Yaskawa INFORM job: sDeep_drilling_(2).JBI

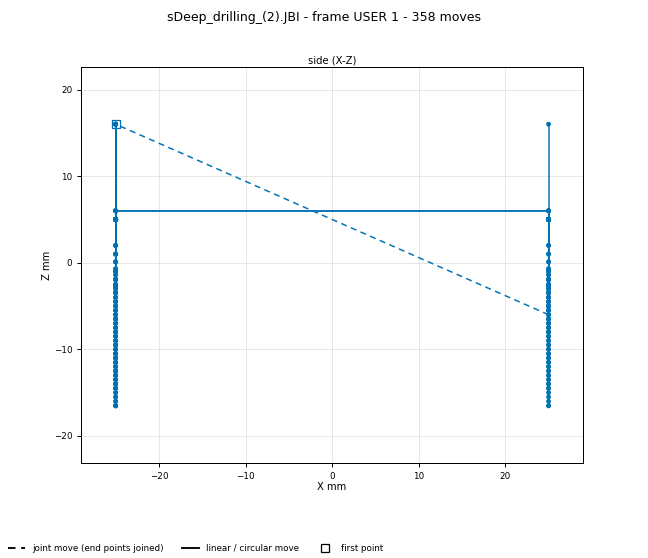
[picture p0: tool path of sDeep_drilling_(2).JBI in frame USER 1, 358 of 358 moves have a stored position in this frame; points joined in program order, loops and branches not executed]
/JOB
//NAME sDeep_drilling_(2)
//POS
///NPOS 194,0,0,0,0,0
///USER 1
///TOOL 3
///POSTYPE USER
///RECTAN
///RCONF 1,0,0,0,0,0
C00000=-25.000,10.000,16.000,0.000,-180.000,-30.000
C00001=-25.000,10.000,16.000,0.000,-180.000,-30.000
C00002=-25.000,10.000,6.000,0.000,-180.000,-30.000
C00003=-25.000,10.000,5.000,0.000,-180.000,-30.000
C00004=-25.000,10.000,-16.535,0.000,-180.000,-30.000
C00005=-25.000,10.000,6.000,0.000,-180.000,-30.000
C00006=25.000,10.000,6.000,0.000,-180.000,-30.000
C00007=25.000,10.000,6.000,0.000,-180.000,-30.000
C00008=25.000,10.000,5.000,0.000,-180.000,-30.000
C00009=25.000,10.000,-16.535,0.000,-180.000,-30.000
C00010=25.000,10.000,6.000,0.000,-180.000,-30.000
C00011=25.000,10.000,16.000,0.000,-180.000,-30.000
C00000=-25.000,10.000,16.000,0.000,-180.000,-30.000
C00001=-25.000,10.000,16.000,0.000,-180.000,-30.000
C00002=-25.000,10.000,6.000,0.000,-180.000,-30.000
C00003=-25.000,10.000,5.000,0.000,-180.000,-30.000
C00004=-25.000,10.000,-16.535,0.000,-180.000,-30.000
C00005=-25.000,10.000,6.000,0.000,-180.000,-30.000
C00006=25.000,10.000,6.000,0.000,-180.000,-30.000
C00007=25.000,10.000,6.000,0.000,-180.000,-30.000
C00008=25.000,10.000,5.000,0.000,-180.000,-30.000
C00009=25.000,10.000,-16.535,0.000,-180.000,-30.000
C00010=25.000,10.000,6.000,0.000,-180.000,-30.000
C00011=25.000,10.000,16.000,0.000,-180.000,-30.000
C00000=-25.000,10.000,16.000,0.000,-180.000,-30.000
C00001=-25.000,10.000,16.000,0.000,-180.000,-30.000
C00002=-25.000,10.000,6.000,0.000,-180.000,-30.000
C00003=-25.000,10.000,5.000,0.000,-180.000,-30.000
C00004=-25.000,10.000,2.000,0.000,-180.000,-30.000
C00005=-25.000,10.000,-1.000,0.000,-180.000,-30.000
C00006=-25.000,10.000,-0.898,0.000,-180.000,-30.000
C00007=-25.000,10.000,-1.900,0.000,-180.000,-30.000
C00008=-25.000,10.000,-1.798,0.000,-180.000,-30.000
C00009=-25.000,10.000,-2.700,0.000,-180.000,-30.000
C00010=-25.000,10.000,-2.598,0.000,-180.000,-30.000
C00011=-25.000,10.000,-3.400,0.000,-180.000,-30.000
C00012=-25.000,10.000,-3.298,0.000,-180.000,-30.000
C00013=-25.000,10.000,-4.000,0.000,-180.000,-30.000
C00014=-25.000,10.000,-3.898,0.000,-180.000,-30.000
C00015=-25.000,10.000,-4.500,0.000,-180.000,-30.000
C00016=-25.000,10.000,-4.398,0.000,-180.000,-30.000
C00017=-25.000,10.000,-5.000,0.000,-180.000,-30.000
C00018=-25.000,10.000,6.000,0.000,-180.000,-30.000
C00019=-25.000,10.000,-3.000,0.000,-180.000,-30.000
C00020=-25.000,10.000,-5.500,0.000,-180.000,-30.000
C00021=-25.000,10.000,-5.398,0.000,-180.000,-30.000
C00022=-25.000,10.000,-6.000,0.000,-180.000,-30.000
C00023=-25.000,10.000,-5.898,0.000,-180.000,-30.000
C00024=-25.000,10.000,-6.500,0.000,-180.000,-30.000
C00025=-25.000,10.000,-6.398,0.000,-180.000,-30.000
C00026=-25.000,10.000,-7.000,0.000,-180.000,-30.000
C00027=-25.000,10.000,-6.898,0.000,-180.000,-30.000
C00028=-25.000,10.000,-7.500,0.000,-180.000,-30.000
C00029=-25.000,10.000,-7.398,0.000,-180.000,-30.000
C00030=-25.000,10.000,-8.000,0.000,-180.000,-30.000
C00031=-25.000,10.000,-7.898,0.000,-180.000,-30.000
C00032=-25.000,10.000,-8.500,0.000,-180.000,-30.000
C00033=-25.000,10.000,-8.398,0.000,-180.000,-30.000
C00034=-25.000,10.000,-9.000,0.000,-180.000,-30.000
C00035=-25.000,10.000,-8.898,0.000,-180.000,-30.000
C00036=-25.000,10.000,-9.500,0.000,-180.000,-30.000
C00037=-25.000,10.000,-9.398,0.000,-180.000,-30.000
C00038=-25.000,10.000,-10.000,0.000,-180.000,-30.000
C00039=-25.000,10.000,6.000,0.000,-180.000,-30.000
C00040=-25.000,10.000,-8.000,0.000,-180.000,-30.000
C00041=-25.000,10.000,-10.500,0.000,-180.000,-30.000
C00042=-25.000,10.000,-10.398,0.000,-180.000,-30.000
C00043=-25.000,10.000,-11.000,0.000,-180.000,-30.000
C00044=-25.000,10.000,-10.898,0.000,-180.000,-30.000
C00045=-25.000,10.000,-11.500,0.000,-180.000,-30.000
C00046=-25.000,10.000,-11.398,0.000,-180.000,-30.000
C00047=-25.000,10.000,-12.000,0.000,-180.000,-30.000
C00048=-25.000,10.000,-11.898,0.000,-180.000,-30.000
C00049=-25.000,10.000,-12.500,0.000,-180.000,-30.000
C00050=-25.000,10.000,-12.398,0.000,-180.000,-30.000
C00051=-25.000,10.000,-13.000,0.000,-180.000,-30.000
C00052=-25.000,10.000,-12.898,0.000,-180.000,-30.000
C00053=-25.000,10.000,-13.500,0.000,-180.000,-30.000
C00054=-25.000,10.000,-13.398,0.000,-180.000,-30.000
C00055=-25.000,10.000,-14.000,0.000,-180.000,-30.000
C00056=-25.000,10.000,-13.898,0.000,-180.000,-30.000
C00057=-25.000,10.000,-14.500,0.000,-180.000,-30.000
C00058=-25.000,10.000,-14.398,0.000,-180.000,-30.000
C00059=-25.000,10.000,-15.000,0.000,-180.000,-30.000
C00060=-25.000,10.000,6.000,0.000,-180.000,-30.000
C00061=-25.000,10.000,-13.000,0.000,-180.000,-30.000
C00062=-25.000,10.000,-15.500,0.000,-180.000,-30.000
C00063=-25.000,10.000,-15.398,0.000,-180.000,-30.000
C00064=-25.000,10.000,-16.000,0.000,-180.000,-30.000
C00065=-25.000,10.000,-15.898,0.000,-180.000,-30.000
C00066=-25.000,10.000,-16.500,0.000,-180.000,-30.000
C00067=-25.000,10.000,-16.398,0.000,-180.000,-30.000
C00068=-25.000,10.000,-16.535,0.000,-180.000,-30.000
C00069=-25.000,10.000,6.000,0.000,-180.000,-30.000
C00070=25.000,10.000,6.000,0.000,-180.000,-30.000
C00071=25.000,10.000,6.000,0.000,-180.000,-30.000
C00072=25.000,10.000,5.000,0.000,-180.000,-30.000
C00073=25.000,10.000,2.000,0.000,-180.000,-30.000
C00074=25.000,10.000,-1.000,0.000,-180.000,-30.000
C00075=25.000,10.000,-0.898,0.000,-180.000,-30.000
C00076=25.000,10.000,-1.900,0.000,-180.000,-30.000
C00077=25.000,10.000,-1.798,0.000,-180.000,-30.000
C00078=25.000,10.000,-2.700,0.000,-180.000,-30.000
C00079=25.000,10.000,-2.598,0.000,-180.000,-30.000
C00080=25.000,10.000,-3.400,0.000,-180.000,-30.000
C00081=25.000,10.000,-3.298,0.000,-180.000,-30.000
C00082=25.000,10.000,-4.000,0.000,-180.000,-30.000
C00083=25.000,10.000,-3.898,0.000,-180.000,-30.000
C00084=25.000,10.000,-4.500,0.000,-180.000,-30.000
C00085=25.000,10.000,-4.398,0.000,-180.000,-30.000
C00086=25.000,10.000,-5.000,0.000,-180.000,-30.000
C00087=25.000,10.000,6.000,0.000,-180.000,-30.000
C00088=25.000,10.000,-3.000,0.000,-180.000,-30.000
C00089=25.000,10.000,-5.500,0.000,-180.000,-30.000
C00090=25.000,10.000,-5.398,0.000,-180.000,-30.000
C00091=25.000,10.000,-6.000,0.000,-180.000,-30.000
C00092=25.000,10.000,-5.898,0.000,-180.000,-30.000
C00093=25.000,10.000,-6.500,0.000,-180.000,-30.000
C00094=25.000,10.000,-6.398,0.000,-180.000,-30.000
C00095=25.000,10.000,-7.000,0.000,-180.000,-30.000
C00096=25.000,10.000,-6.898,0.000,-180.000,-30.000
C00097=25.000,10.000,-7.500,0.000,-180.000,-30.000
C00098=25.000,10.000,-7.398,0.000,-180.000,-30.000
C00099=25.000,10.000,-8.000,0.000,-180.000,-30.000
C00100=25.000,10.000,-7.898,0.000,-180.000,-30.000
C00101=25.000,10.000,-8.500,0.000,-180.000,-30.000
C00102=25.000,10.000,-8.398,0.000,-180.000,-30.000
C00103=25.000,10.000,-9.000,0.000,-180.000,-30.000
C00104=25.000,10.000,-8.898,0.000,-180.000,-30.000
C00105=25.000,10.000,-9.500,0.000,-180.000,-30.000
C00106=25.000,10.000,-9.398,0.000,-180.000,-30.000
C00107=25.000,10.000,-10.000,0.000,-180.000,-30.000
C00108=25.000,10.000,6.000,0.000,-180.000,-30.000
C00109=25.000,10.000,-8.000,0.000,-180.000,-30.000
C00110=25.000,10.000,-10.500,0.000,-180.000,-30.000
C00111=25.000,10.000,-10.398,0.000,-180.000,-30.000
C00112=25.000,10.000,-11.000,0.000,-180.000,-30.000
C00113=25.000,10.000,-10.898,0.000,-180.000,-30.000
C00114=25.000,10.000,-11.500,0.000,-180.000,-30.000
C00115=25.000,10.000,-11.398,0.000,-180.000,-30.000
C00116=25.000,10.000,-12.000,0.000,-180.000,-30.000
C00117=25.000,10.000,-11.898,0.000,-180.000,-30.000
C00118=25.000,10.000,-12.500,0.000,-180.000,-30.000
C00119=25.000,10.000,-12.398,0.000,-180.000,-30.000
C00120=25.000,10.000,-13.000,0.000,-180.000,-30.000
C00121=25.000,10.000,-12.898,0.000,-180.000,-30.000
C00122=25.000,10.000,-13.500,0.000,-180.000,-30.000
C00123=25.000,10.000,-13.398,0.000,-180.000,-30.000
C00124=25.000,10.000,-14.000,0.000,-180.000,-30.000
C00125=25.000,10.000,-13.898,0.000,-180.000,-30.000
C00126=25.000,10.000,-14.500,0.000,-180.000,-30.000
C00127=25.000,10.000,-14.398,0.000,-180.000,-30.000
C00128=25.000,10.000,-15.000,0.000,-180.000,-30.000
C00129=25.000,10.000,6.000,0.000,-180.000,-30.000
C00130=25.000,10.000,-13.000,0.000,-180.000,-30.000
C00131=25.000,10.000,-15.500,0.000,-180.000,-30.000
C00132=25.000,10.000,-15.398,0.000,-180.000,-30.000
C00133=25.000,10.000,-16.000,0.000,-180.000,-30.000
C00134=25.000,10.000,-15.898,0.000,-180.000,-30.000
C00135=25.000,10.000,-16.500,0.000,-180.000,-30.000
C00136=25.000,10.000,-16.398,0.000,-180.000,-30.000
C00137=25.000,10.000,-16.535,0.000,-180.000,-30.000
C00138=25.000,10.000,6.000,0.000,-180.000,-30.000
C00139=25.000,10.000,16.000,0.000,-180.000,-30.000
C00000=-25.000,10.000,16.000,0.000,-180.000,-30.000
C00001=-25.000,10.000,16.000,0.000,-180.000,-30.000
C00002=-25.000,10.000,6.000,0.000,-180.000,-30.000
C00003=-25.000,10.000,5.000,0.000,-180.000,-30.000
C00004=-25.000,10.000,2.000,0.000,-180.000,-30.000
C00005=-25.000,10.000,-1.000,0.000,-180.000,-30.000
C00006=-25.000,10.000,5.000,0.000,-180.000,-30.000
C00007=-25.000,10.000,1.000,0.000,-180.000,-30.000
C00008=-25.000,10.000,-1.900,0.000,-180.000,-30.000
C00009=-25.000,10.000,5.000,0.000,-180.000,-30.000
C00010=-25.000,10.000,0.100,0.000,-180.000,-30.000
C00011=-25.000,10.000,-2.700,0.000,-180.000,-30.000
C00012=-25.000,10.000,5.000,0.000,-180.000,-30.000
C00013=-25.000,10.000,-0.700,0.000,-180.000,-30.000
C00014=-25.000,10.000,-3.400,0.000,-180.000,-30.000
C00015=-25.000,10.000,5.000,0.000,-180.000,-30.000
C00016=-25.000,10.000,-1.400,0.000,-180.000,-30.000
C00017=-25.000,10.000,-4.000,0.000,-180.000,-30.000
C00018=-25.000,10.000,5.000,0.000,-180.000,-30.000
C00019=-25.000,10.000,-2.000,0.000,-180.000,-30.000
C00020=-25.000,10.000,-4.500,0.000,-180.000,-30.000
C00021=-25.000,10.000,5.000,0.000,-180.000,-30.000
C00022=-25.000,10.000,-2.500,0.000,-180.000,-30.000
C00023=-25.000,10.000,-5.000,0.000,-180.000,-30.000
C00024=-25.000,10.000,5.000,0.000,-180.000,-30.000
C00025=-25.000,10.000,-3.000,0.000,-180.000,-30.000
C00026=-25.000,10.000,-5.500,0.000,-180.000,-30.000
C00027=-25.000,10.000,5.000,0.000,-180.000,-30.000
C00028=-25.000,10.000,-3.500,0.000,-180.000,-30.000
C00029=-25.000,10.000,-6.000,0.000,-180.000,-30.000
C00030=-25.000,10.000,5.000,0.000,-180.000,-30.000
C00031=-25.000,10.000,-4.000,0.000,-180.000,-30.000
C00032=-25.000,10.000,-6.500,0.000,-180.000,-30.000
C00033=-25.000,10.000,5.000,0.000,-180.000,-30.000
C00034=-25.000,10.000,-4.500,0.000,-180.000,-30.000
C00035=-25.000,10.000,-7.000,0.000,-180.000,-30.000
C00036=-25.000,10.000,5.000,0.000,-180.000,-30.000
C00037=-25.000,10.000,-5.000,0.000,-180.000,-30.000
C00038=-25.000,10.000,-7.500,0.000,-180.000,-30.000
C00039=-25.000,10.000,5.000,0.000,-180.000,-30.000
C00040=-25.000,10.000,-5.500,0.000,-180.000,-30.000
C00041=-25.000,10.000,-8.000,0.000,-180.000,-30.000
C00042=-25.000,10.000,5.000,0.000,-180.000,-30.000
C00043=-25.000,10.000,-6.000,0.000,-180.000,-30.000
C00044=-25.000,10.000,-8.500,0.000,-180.000,-30.000
C00045=-25.000,10.000,5.000,0.000,-180.000,-30.000
C00046=-25.000,10.000,-6.500,0.000,-180.000,-30.000
C00047=-25.000,10.000,-9.000,0.000,-180.000,-30.000
C00048=-25.000,10.000,5.000,0.000,-180.000,-30.000
C00049=-25.000,10.000,-7.000,0.000,-180.000,-30.000
C00050=-25.000,10.000,-9.500,0.000,-180.000,-30.000
C00051=-25.000,10.000,5.000,0.000,-180.000,-30.000
C00052=-25.000,10.000,-7.500,0.000,-180.000,-30.000
C00053=-25.000,10.000,-10.000,0.000,-180.000,-30.000
C00054=-25.000,10.000,5.000,0.000,-180.000,-30.000
C00055=-25.000,10.000,-8.000,0.000,-180.000,-30.000
C00056=-25.000,10.000,-10.500,0.000,-180.000,-30.000
C00057=-25.000,10.000,5.000,0.000,-180.000,-30.000
C00058=-25.000,10.000,-8.500,0.000,-180.000,-30.000
C00059=-25.000,10.000,-11.000,0.000,-180.000,-30.000
C00060=-25.000,10.000,5.000,0.000,-180.000,-30.000
C00061=-25.000,10.000,-9.000,0.000,-180.000,-30.000
C00062=-25.000,10.000,-11.500,0.000,-180.000,-30.000
C00063=-25.000,10.000,5.000,0.000,-180.000,-30.000
C00064=-25.000,10.000,-9.500,0.000,-180.000,-30.000
C00065=-25.000,10.000,-12.000,0.000,-180.000,-30.000
C00066=-25.000,10.000,5.000,0.000,-180.000,-30.000
C00067=-25.000,10.000,-10.000,0.000,-180.000,-30.000
C00068=-25.000,10.000,-12.500,0.000,-180.000,-30.000
C00069=-25.000,10.000,5.000,0.000,-180.000,-30.000
C00070=-25.000,10.000,-10.500,0.000,-180.000,-30.000
C00071=-25.000,10.000,-13.000,0.000,-180.000,-30.000
C00072=-25.000,10.000,5.000,0.000,-180.000,-30.000
C00073=-25.000,10.000,-11.000,0.000,-180.000,-30.000
C00074=-25.000,10.000,-13.500,0.000,-180.000,-30.000
C00075=-25.000,10.000,5.000,0.000,-180.000,-30.000
C00076=-25.000,10.000,-11.500,0.000,-180.000,-30.000
C00077=-25.000,10.000,-14.000,0.000,-180.000,-30.000
C00078=-25.000,10.000,5.000,0.000,-180.000,-30.000
C00079=-25.000,10.000,-12.000,0.000,-180.000,-30.000
C00080=-25.000,10.000,-14.500,0.000,-180.000,-30.000
C00081=-25.000,10.000,5.000,0.000,-180.000,-30.000
C00082=-25.000,10.000,-12.500,0.000,-180.000,-30.000
C00083=-25.000,10.000,-15.000,0.000,-180.000,-30.000
C00084=-25.000,10.000,5.000,0.000,-180.000,-30.000
C00085=-25.000,10.000,-13.000,0.000,-180.000,-30.000
C00086=-25.000,10.000,-15.500,0.000,-180.000,-30.000
C00087=-25.000,10.000,5.000,0.000,-180.000,-30.000
C00088=-25.000,10.000,-13.500,0.000,-180.000,-30.000
C00089=-25.000,10.000,-16.000,0.000,-180.000,-30.000
C00090=-25.000,10.000,5.000,0.000,-180.000,-30.000
C00091=-25.000,10.000,-14.000,0.000,-180.000,-30.000
C00092=-25.000,10.000,-16.500,0.000,-180.000,-30.000
C00093=-25.000,10.000,5.000,0.000,-180.000,-30.000
C00094=-25.000,10.000,-14.500,0.000,-180.000,-30.000
C00095=-25.000,10.000,-16.535,0.000,-180.000,-30.000
C00096=-25.000,10.000,6.000,0.000,-180.000,-30.000
C00097=25.000,10.000,6.000,0.000,-180.000,-30.000
C00098=25.000,10.000,6.000,0.000,-180.000,-30.000
C00099=25.000,10.000,5.000,0.000,-180.000,-30.000
C00100=25.000,10.000,2.000,0.000,-180.000,-30.000
C00101=25.000,10.000,-1.000,0.000,-180.000,-30.000
C00102=25.000,10.000,5.000,0.000,-180.000,-30.000
C00103=25.000,10.000,1.000,0.000,-180.000,-30.000
C00104=25.000,10.000,-1.900,0.000,-180.000,-30.000
C00105=25.000,10.000,5.000,0.000,-180.000,-30.000
C00106=25.000,10.000,0.100,0.000,-180.000,-30.000
C00107=25.000,10.000,-2.700,0.000,-180.000,-30.000
C00108=25.000,10.000,5.000,0.000,-180.000,-30.000
C00109=25.000,10.000,-0.700,0.000,-180.000,-30.000
C00110=25.000,10.000,-3.400,0.000,-180.000,-30.000
C00111=25.000,10.000,5.000,0.000,-180.000,-30.000
C00112=25.000,10.000,-1.400,0.000,-180.000,-30.000
C00113=25.000,10.000,-4.000,0.000,-180.000,-30.000
C00114=25.000,10.000,5.000,0.000,-180.000,-30.000
C00115=25.000,10.000,-2.000,0.000,-180.000,-30.000
C00116=25.000,10.000,-4.500,0.000,-180.000,-30.000
C00117=25.000,10.000,5.000,0.000,-180.000,-30.000
C00118=25.000,10.000,-2.500,0.000,-180.000,-30.000
C00119=25.000,10.000,-5.000,0.000,-180.000,-30.000
C00120=25.000,10.000,5.000,0.000,-180.000,-30.000
C00121=25.000,10.000,-3.000,0.000,-180.000,-30.000
C00122=25.000,10.000,-5.500,0.000,-180.000,-30.000
C00123=25.000,10.000,5.000,0.000,-180.000,-30.000
C00124=25.000,10.000,-3.500,0.000,-180.000,-30.000
C00125=25.000,10.000,-6.000,0.000,-180.000,-30.000
C00126=25.000,10.000,5.000,0.000,-180.000,-30.000
C00127=25.000,10.000,-4.000,0.000,-180.000,-30.000
C00128=25.000,10.000,-6.500,0.000,-180.000,-30.000
C00129=25.000,10.000,5.000,0.000,-180.000,-30.000
C00130=25.000,10.000,-4.500,0.000,-180.000,-30.000
C00131=25.000,10.000,-7.000,0.000,-180.000,-30.000
C00132=25.000,10.000,5.000,0.000,-180.000,-30.000
C00133=25.000,10.000,-5.000,0.000,-180.000,-30.000
C00134=25.000,10.000,-7.500,0.000,-180.000,-30.000
C00135=25.000,10.000,5.000,0.000,-180.000,-30.000
C00136=25.000,10.000,-5.500,0.000,-180.000,-30.000
C00137=25.000,10.000,-8.000,0.000,-180.000,-30.000
C00138=25.000,10.000,5.000,0.000,-180.000,-30.000
C00139=25.000,10.000,-6.000,0.000,-180.000,-30.000
C00140=25.000,10.000,-8.500,0.000,-180.000,-30.000
C00141=25.000,10.000,5.000,0.000,-180.000,-30.000
C00142=25.000,10.000,-6.500,0.000,-180.000,-30.000
C00143=25.000,10.000,-9.000,0.000,-180.000,-30.000
C00144=25.000,10.000,5.000,0.000,-180.000,-30.000
C00145=25.000,10.000,-7.000,0.000,-180.000,-30.000
C00146=25.000,10.000,-9.500,0.000,-180.000,-30.000
C00147=25.000,10.000,5.000,0.000,-180.000,-30.000
C00148=25.000,10.000,-7.500,0.000,-180.000,-30.000
C00149=25.000,10.000,-10.000,0.000,-180.000,-30.000
C00150=25.000,10.000,5.000,0.000,-180.000,-30.000
C00151=25.000,10.000,-8.000,0.000,-180.000,-30.000
C00152=25.000,10.000,-10.500,0.000,-180.000,-30.000
C00153=25.000,10.000,5.000,0.000,-180.000,-30.000
C00154=25.000,10.000,-8.500,0.000,-180.000,-30.000
C00155=25.000,10.000,-11.000,0.000,-180.000,-30.000
C00156=25.000,10.000,5.000,0.000,-180.000,-30.000
C00157=25.000,10.000,-9.000,0.000,-180.000,-30.000
C00158=25.000,10.000,-11.500,0.000,-180.000,-30.000
C00159=25.000,10.000,5.000,0.000,-180.000,-30.000
C00160=25.000,10.000,-9.500,0.000,-180.000,-30.000
C00161=25.000,10.000,-12.000,0.000,-180.000,-30.000
C00162=25.000,10.000,5.000,0.000,-180.000,-30.000
C00163=25.000,10.000,-10.000,0.000,-180.000,-30.000
C00164=25.000,10.000,-12.500,0.000,-180.000,-30.000
C00165=25.000,10.000,5.000,0.000,-180.000,-30.000
C00166=25.000,10.000,-10.500,0.000,-180.000,-30.000
C00167=25.000,10.000,-13.000,0.000,-180.000,-30.000
C00168=25.000,10.000,5.000,0.000,-180.000,-30.000
C00169=25.000,10.000,-11.000,0.000,-180.000,-30.000
C00170=25.000,10.000,-13.500,0.000,-180.000,-30.000
C00171=25.000,10.000,5.000,0.000,-180.000,-30.000
C00172=25.000,10.000,-11.500,0.000,-180.000,-30.000
C00173=25.000,10.000,-14.000,0.000,-180.000,-30.000
C00174=25.000,10.000,5.000,0.000,-180.000,-30.000
C00175=25.000,10.000,-12.000,0.000,-180.000,-30.000
C00176=25.000,10.000,-14.500,0.000,-180.000,-30.000
C00177=25.000,10.000,5.000,0.000,-180.000,-30.000
C00178=25.000,10.000,-12.500,0.000,-180.000,-30.000
C00179=25.000,10.000,-15.000,0.000,-180.000,-30.000
C00180=25.000,10.000,5.000,0.000,-180.000,-30.000
C00181=25.000,10.000,-13.000,0.000,-180.000,-30.000
C00182=25.000,10.000,-15.500,0.000,-180.000,-30.000
C00183=25.000,10.000,5.000,0.000,-180.000,-30.000
C00184=25.000,10.000,-13.500,0.000,-180.000,-30.000
C00185=25.000,10.000,-16.000,0.000,-180.000,-30.000
C00186=25.000,10.000,5.000,0.000,-180.000,-30.000
C00187=25.000,10.000,-14.000,0.000,-180.000,-30.000
C00188=25.000,10.000,-16.500,0.000,-180.000,-30.000
C00189=25.000,10.000,5.000,0.000,-180.000,-30.000
C00190=25.000,10.000,-14.500,0.000,-180.000,-30.000
C00191=25.000,10.000,-16.535,0.000,-180.000,-30.000
C00192=25.000,10.000,6.000,0.000,-180.000,-30.000
C00193=25.000,10.000,16.000,0.000,-180.000,-30.000
//INST
///ATTR SC,RW,RJ
////FRAME USER 1
///GROUP1 RB1
///LVARS 2,0,0,0,0,0,0,0
NOP
SET LB000 1
SET LB001 25
MOVJ C00000 VJ=17
' Cutting Move Starts
MOVL C00001 V=17 PL=LB000 ACC=LB001 DEC=LB001
MOVL C00002 V=17 PL=LB000 ACC=LB001 DEC=LB001
MOVL C00003 V=17 PL=LB000 ACC=LB001 DEC=LB001
MOVL C00004 V=7 PL=LB000 ACC=LB001 DEC=LB001
MOVL C00005 V=17 PL=LB000 ACC=LB001 DEC=LB001
MOVL C00006 V=17 PL=LB000 ACC=LB001 DEC=LB001
MOVL C00007 V=17 PL=LB000 ACC=LB001 DEC=LB001
MOVL C00008 V=17 PL=LB000 ACC=LB001 DEC=LB001
MOVL C00009 V=7 PL=LB000 ACC=LB001 DEC=LB001
MOVL C00010 V=17 PL=LB000 ACC=LB001 DEC=LB001
' Rapid Move Starts
MOVL C00011 V=17 PL=LB000 ACC=LB001 DEC=LB001
' By Autodesk Fusion CAM 2.0.20494
' Tool = 3
' Spindle = 5000 RPM
' Set Position Level
' Set Acceleration
' Program Start
' First Toolpath Point
' Last Toolpath Point
MOVJ C00000 VJ=17
' Cutting Move Starts
MOVL C00001 V=17 PL=LB000 ACC=LB001 DEC=LB001
MOVL C00002 V=17 PL=LB000 ACC=LB001 DEC=LB001
MOVL C00003 V=17 PL=LB000 ACC=LB001 DEC=LB001
MOVL C00004 V=7 PL=LB000 ACC=LB001 DEC=LB001
MOVL C00005 V=17 PL=LB000 ACC=LB001 DEC=LB001
MOVL C00006 V=17 PL=LB000 ACC=LB001 DEC=LB001
MOVL C00007 V=17 PL=LB000 ACC=LB001 DEC=LB001
MOVL C00008 V=17 PL=LB000 ACC=LB001 DEC=LB001
MOVL C00009 V=7 PL=LB000 ACC=LB001 DEC=LB001
MOVL C00010 V=17 PL=LB000 ACC=LB001 DEC=LB001
' Rapid Move Starts
MOVL C00011 V=17 PL=LB000 ACC=LB001 DEC=LB001
' By Autodesk Fusion CAM 2.0.20494
' Tool = 3
' Spindle = 5000 RPM
' Set Position Level
' Set Acceleration
' Program Start
' First Toolpath Point
' Last Toolpath Point
MOVJ C00000 VJ=17
' Cutting Move Starts
MOVL C00001 V=17 PL=LB000 ACC=LB001 DEC=LB001
MOVL C00002 V=17 PL=LB000 ACC=LB001 DEC=LB001
MOVL C00003 V=17 PL=LB000 ACC=LB001 DEC=LB001
MOVL C00004 V=17 PL=LB000 ACC=LB001 DEC=LB001
MOVL C00005 V=7 PL=LB000 ACC=LB001 DEC=LB001
MOVL C00006 V=17 PL=LB000 ACC=LB001 DEC=LB001
MOVL C00007 V=7 PL=LB000 ACC=LB001 DEC=LB001
MOVL C00008 V=17 PL=LB000 ACC=LB001 DEC=LB001
MOVL C00009 V=7 PL=LB000 ACC=LB001 DEC=LB001
MOVL C00010 V=17 PL=LB000 ACC=LB001 DEC=LB001
MOVL C00011 V=7 PL=LB000 ACC=LB001 DEC=LB001
MOVL C00012 V=17 PL=LB000 ACC=LB001 DEC=LB001
MOVL C00013 V=7 PL=LB000 ACC=LB001 DEC=LB001
MOVL C00014 V=17 PL=LB000 ACC=LB001 DEC=LB001
MOVL C00015 V=7 PL=LB000 ACC=LB001 DEC=LB001
MOVL C00016 V=17 PL=LB000 ACC=LB001 DEC=LB001
MOVL C00017 V=7 PL=LB000 ACC=LB001 DEC=LB001
MOVL C00018 V=17 PL=LB000 ACC=LB001 DEC=LB001
MOVL C00019 V=17 PL=LB000 ACC=LB001 DEC=LB001
MOVL C00020 V=7 PL=LB000 ACC=LB001 DEC=LB001
MOVL C00021 V=17 PL=LB000 ACC=LB001 DEC=LB001
MOVL C00022 V=7 PL=LB000 ACC=LB001 DEC=LB001
MOVL C00023 V=17 PL=LB000 ACC=LB001 DEC=LB001
MOVL C00024 V=7 PL=LB000 ACC=LB001 DEC=LB001
MOVL C00025 V=17 PL=LB000 ACC=LB001 DEC=LB001
MOVL C00026 V=7 PL=LB000 ACC=LB001 DEC=LB001
MOVL C00027 V=17 PL=LB000 ACC=LB001 DEC=LB001
MOVL C00028 V=7 PL=LB000 ACC=LB001 DEC=LB001
MOVL C00029 V=17 PL=LB000 ACC=LB001 DEC=LB001
MOVL C00030 V=7 PL=LB000 ACC=LB001 DEC=LB001
MOVL C00031 V=17 PL=LB000 ACC=LB001 DEC=LB001
MOVL C00032 V=7 PL=LB000 ACC=LB001 DEC=LB001
MOVL C00033 V=17 PL=LB000 ACC=LB001 DEC=LB001
MOVL C00034 V=7 PL=LB000 ACC=LB001 DEC=LB001
MOVL C00035 V=17 PL=LB000 ACC=LB001 DEC=LB001
MOVL C00036 V=7 PL=LB000 ACC=LB001 DEC=LB001
MOVL C00037 V=17 PL=LB000 ACC=LB001 DEC=LB001
MOVL C00038 V=7 PL=LB000 ACC=LB001 DEC=LB001
MOVL C00039 V=17 PL=LB000 ACC=LB001 DEC=LB001
MOVL C00040 V=17 PL=LB000 ACC=LB001 DEC=LB001
MOVL C00041 V=7 PL=LB000 ACC=LB001 DEC=LB001
MOVL C00042 V=17 PL=LB000 ACC=LB001 DEC=LB001
MOVL C00043 V=7 PL=LB000 ACC=LB001 DEC=LB001
MOVL C00044 V=17 PL=LB000 ACC=LB001 DEC=LB001
MOVL C00045 V=7 PL=LB000 ACC=LB001 DEC=LB001
MOVL C00046 V=17 PL=LB000 ACC=LB001 DEC=LB001
MOVL C00047 V=7 PL=LB000 ACC=LB001 DEC=LB001
MOVL C00048 V=17 PL=LB000 ACC=LB001 DEC=LB001
MOVL C00049 V=7 PL=LB000 ACC=LB001 DEC=LB001
MOVL C00050 V=17 PL=LB000 ACC=LB001 DEC=LB001
MOVL C00051 V=7 PL=LB000 ACC=LB001 DEC=LB001
MOVL C00052 V=17 PL=LB000 ACC=LB001 DEC=LB001
MOVL C00053 V=7 PL=LB000 ACC=LB001 DEC=LB001
MOVL C00054 V=17 PL=LB000 ACC=LB001 DEC=LB001
MOVL C00055 V=7 PL=LB000 ACC=LB001 DEC=LB001
MOVL C00056 V=17 PL=LB000 ACC=LB001 DEC=LB001
MOVL C00057 V=7 PL=LB000 ACC=LB001 DEC=LB001
MOVL C00058 V=17 PL=LB000 ACC=LB001 DEC=LB001
MOVL C00059 V=7 PL=LB000 ACC=LB001 DEC=LB001
MOVL C00060 V=17 PL=LB000 ACC=LB001 DEC=LB001
MOVL C00061 V=17 PL=LB000 ACC=LB001 DEC=LB001
MOVL C00062 V=7 PL=LB000 ACC=LB001 DEC=LB001
MOVL C00063 V=17 PL=LB000 ACC=LB001 DEC=LB001
MOVL C00064 V=7 PL=LB000 ACC=LB001 DEC=LB001
MOVL C00065 V=17 PL=LB000 ACC=LB001 DEC=LB001
MOVL C00066 V=7 PL=LB000 ACC=LB001 DEC=LB001
MOVL C00067 V=17 PL=LB000 ACC=LB001 DEC=LB001
MOVL C00068 V=7 PL=LB000 ACC=LB001 DEC=LB001
MOVL C00069 V=17 PL=LB000 ACC=LB001 DEC=LB001
MOVL C00070 V=17 PL=LB000 ACC=LB001 DEC=LB001
MOVL C00071 V=17 PL=LB000 ACC=LB001 DEC=LB001
MOVL C00072 V=17 PL=LB000 ACC=LB001 DEC=LB001
MOVL C00073 V=17 PL=LB000 ACC=LB001 DEC=LB001
MOVL C00074 V=7 PL=LB000 ACC=LB001 DEC=LB001
MOVL C00075 V=17 PL=LB000 ACC=LB001 DEC=LB001
MOVL C00076 V=7 PL=LB000 ACC=LB001 DEC=LB001
MOVL C00077 V=17 PL=LB000 ACC=LB001 DEC=LB001
MOVL C00078 V=7 PL=LB000 ACC=LB001 DEC=LB001
MOVL C00079 V=17 PL=LB000 ACC=LB001 DEC=LB001
MOVL C00080 V=7 PL=LB000 ACC=LB001 DEC=LB001
MOVL C00081 V=17 PL=LB000 ACC=LB001 DEC=LB001
MOVL C00082 V=7 PL=LB000 ACC=LB001 DEC=LB001
MOVL C00083 V=17 PL=LB000 ACC=LB001 DEC=LB001
MOVL C00084 V=7 PL=LB000 ACC=LB001 DEC=LB001
MOVL C00085 V=17 PL=LB000 ACC=LB001 DEC=LB001
MOVL C00086 V=7 PL=LB000 ACC=LB001 DEC=LB001
MOVL C00087 V=17 PL=LB000 ACC=LB001 DEC=LB001
MOVL C00088 V=17 PL=LB000 ACC=LB001 DEC=LB001
MOVL C00089 V=7 PL=LB000 ACC=LB001 DEC=LB001
MOVL C00090 V=17 PL=LB000 ACC=LB001 DEC=LB001
MOVL C00091 V=7 PL=LB000 ACC=LB001 DEC=LB001
MOVL C00092 V=17 PL=LB000 ACC=LB001 DEC=LB001
MOVL C00093 V=7 PL=LB000 ACC=LB001 DEC=LB001
MOVL C00094 V=17 PL=LB000 ACC=LB001 DEC=LB001
MOVL C00095 V=7 PL=LB000 ACC=LB001 DEC=LB001
MOVL C00096 V=17 PL=LB000 ACC=LB001 DEC=LB001
MOVL C00097 V=7 PL=LB000 ACC=LB001 DEC=LB001
MOVL C00098 V=17 PL=LB000 ACC=LB001 DEC=LB001
MOVL C00099 V=7 PL=LB000 ACC=LB001 DEC=LB001
MOVL C00100 V=17 PL=LB000 ACC=LB001 DEC=LB001
MOVL C00101 V=7 PL=LB000 ACC=LB001 DEC=LB001
MOVL C00102 V=17 PL=LB000 ACC=LB001 DEC=LB001
MOVL C00103 V=7 PL=LB000 ACC=LB001 DEC=LB001
MOVL C00104 V=17 PL=LB000 ACC=LB001 DEC=LB001
MOVL C00105 V=7 PL=LB000 ACC=LB001 DEC=LB001
MOVL C00106 V=17 PL=LB000 ACC=LB001 DEC=LB001
MOVL C00107 V=7 PL=LB000 ACC=LB001 DEC=LB001
MOVL C00108 V=17 PL=LB000 ACC=LB001 DEC=LB001
MOVL C00109 V=17 PL=LB000 ACC=LB001 DEC=LB001
MOVL C00110 V=7 PL=LB000 ACC=LB001 DEC=LB001
MOVL C00111 V=17 PL=LB000 ACC=LB001 DEC=LB001
MOVL C00112 V=7 PL=LB000 ACC=LB001 DEC=LB001
MOVL C00113 V=17 PL=LB000 ACC=LB001 DEC=LB001
MOVL C00114 V=7 PL=LB000 ACC=LB001 DEC=LB001
MOVL C00115 V=17 PL=LB000 ACC=LB001 DEC=LB001
MOVL C00116 V=7 PL=LB000 ACC=LB001 DEC=LB001
MOVL C00117 V=17 PL=LB000 ACC=LB001 DEC=LB001
MOVL C00118 V=7 PL=LB000 ACC=LB001 DEC=LB001
MOVL C00119 V=17 PL=LB000 ACC=LB001 DEC=LB001
MOVL C00120 V=7 PL=LB000 ACC=LB001 DEC=LB001
MOVL C00121 V=17 PL=LB000 ACC=LB001 DEC=LB001
MOVL C00122 V=7 PL=LB000 ACC=LB001 DEC=LB001
MOVL C00123 V=17 PL=LB000 ACC=LB001 DEC=LB001
MOVL C00124 V=7 PL=LB000 ACC=LB001 DEC=LB001
MOVL C00125 V=17 PL=LB000 ACC=LB001 DEC=LB001
MOVL C00126 V=7 PL=LB000 ACC=LB001 DEC=LB001
MOVL C00127 V=17 PL=LB000 ACC=LB001 DEC=LB001
MOVL C00128 V=7 PL=LB000 ACC=LB001 DEC=LB001
MOVL C00129 V=17 PL=LB000 ACC=LB001 DEC=LB001
MOVL C00130 V=17 PL=LB000 ACC=LB001 DEC=LB001
MOVL C00131 V=7 PL=LB000 ACC=LB001 DEC=LB001
MOVL C00132 V=17 PL=LB000 ACC=LB001 DEC=LB001
MOVL C00133 V=7 PL=LB000 ACC=LB001 DEC=LB001
MOVL C00134 V=17 PL=LB000 ACC=LB001 DEC=LB001
MOVL C00135 V=7 PL=LB000 ACC=LB001 DEC=LB001
MOVL C00136 V=17 PL=LB000 ACC=LB001 DEC=LB001
MOVL C00137 V=7 PL=LB000 ACC=LB001 DEC=LB001
MOVL C00138 V=17 PL=LB000 ACC=LB001 DEC=LB001
' Rapid Move Starts
MOVL C00139 V=17 PL=LB000 ACC=LB001 DEC=LB001
' By Autodesk Fusion CAM 2.0.20494
' Tool = 3
' Spindle = 5000 RPM
' Set Position Level
' Set Acceleration
' Program Start
' First Toolpath Point
' Last Toolpath Point
MOVJ C00000 VJ=17
' Cutting Move Starts
MOVL C00001 V=17 PL=LB000 ACC=LB001 DEC=LB001
MOVL C00002 V=17 PL=LB000 ACC=LB001 DEC=LB001
MOVL C00003 V=17 PL=LB000 ACC=LB001 DEC=LB001
MOVL C00004 V=17 PL=LB000 ACC=LB001 DEC=LB001
MOVL C00005 V=7 PL=LB000 ACC=LB001 DEC=LB001
MOVL C00006 V=17 PL=LB000 ACC=LB001 DEC=LB001
MOVL C00007 V=17 PL=LB000 ACC=LB001 DEC=LB001
MOVL C00008 V=7 PL=LB000 ACC=LB001 DEC=LB001
MOVL C00009 V=17 PL=LB000 ACC=LB001 DEC=LB001
MOVL C00010 V=17 PL=LB000 ACC=LB001 DEC=LB001
MOVL C00011 V=7 PL=LB000 ACC=LB001 DEC=LB001
MOVL C00012 V=17 PL=LB000 ACC=LB001 DEC=LB001
MOVL C00013 V=17 PL=LB000 ACC=LB001 DEC=LB001
MOVL C00014 V=7 PL=LB000 ACC=LB001 DEC=LB001
MOVL C00015 V=17 PL=LB000 ACC=LB001 DEC=LB001
MOVL C00016 V=17 PL=LB000 ACC=LB001 DEC=LB001
MOVL C00017 V=7 PL=LB000 ACC=LB001 DEC=LB001
MOVL C00018 V=17 PL=LB000 ACC=LB001 DEC=LB001
MOVL C00019 V=17 PL=LB000 ACC=LB001 DEC=LB001
MOVL C00020 V=7 PL=LB000 ACC=LB001 DEC=LB001
MOVL C00021 V=17 PL=LB000 ACC=LB001 DEC=LB001
MOVL C00022 V=17 PL=LB000 ACC=LB001 DEC=LB001
MOVL C00023 V=7 PL=LB000 ACC=LB001 DEC=LB001
MOVL C00024 V=17 PL=LB000 ACC=LB001 DEC=LB001
MOVL C00025 V=17 PL=LB000 ACC=LB001 DEC=LB001
MOVL C00026 V=7 PL=LB000 ACC=LB001 DEC=LB001
MOVL C00027 V=17 PL=LB000 ACC=LB001 DEC=LB001
MOVL C00028 V=17 PL=LB000 ACC=LB001 DEC=LB001
MOVL C00029 V=7 PL=LB000 ACC=LB001 DEC=LB001
MOVL C00030 V=17 PL=LB000 ACC=LB001 DEC=LB001
MOVL C00031 V=17 PL=LB000 ACC=LB001 DEC=LB001
MOVL C00032 V=7 PL=LB000 ACC=LB001 DEC=LB001
MOVL C00033 V=17 PL=LB000 ACC=LB001 DEC=LB001
MOVL C00034 V=17 PL=LB000 ACC=LB001 DEC=LB001
MOVL C00035 V=7 PL=LB000 ACC=LB001 DEC=LB001
MOVL C00036 V=17 PL=LB000 ACC=LB001 DEC=LB001
MOVL C00037 V=17 PL=LB000 ACC=LB001 DEC=LB001
MOVL C00038 V=7 PL=LB000 ACC=LB001 DEC=LB001
MOVL C00039 V=17 PL=LB000 ACC=LB001 DEC=LB001
MOVL C00040 V=17 PL=LB000 ACC=LB001 DEC=LB001
MOVL C00041 V=7 PL=LB000 ACC=LB001 DEC=LB001
MOVL C00042 V=17 PL=LB000 ACC=LB001 DEC=LB001
MOVL C00043 V=17 PL=LB000 ACC=LB001 DEC=LB001
MOVL C00044 V=7 PL=LB000 ACC=LB001 DEC=LB001
MOVL C00045 V=17 PL=LB000 ACC=LB001 DEC=LB001
MOVL C00046 V=17 PL=LB000 ACC=LB001 DEC=LB001
MOVL C00047 V=7 PL=LB000 ACC=LB001 DEC=LB001
MOVL C00048 V=17 PL=LB000 ACC=LB001 DEC=LB001
MOVL C00049 V=17 PL=LB000 ACC=LB001 DEC=LB001
MOVL C00050 V=7 PL=LB000 ACC=LB001 DEC=LB001
MOVL C00051 V=17 PL=LB000 ACC=LB001 DEC=LB001
MOVL C00052 V=17 PL=LB000 ACC=LB001 DEC=LB001
MOVL C00053 V=7 PL=LB000 ACC=LB001 DEC=LB001
MOVL C00054 V=17 PL=LB000 ACC=LB001 DEC=LB001
MOVL C00055 V=17 PL=LB000 ACC=LB001 DEC=LB001
MOVL C00056 V=7 PL=LB000 ACC=LB001 DEC=LB001
MOVL C00057 V=17 PL=LB000 ACC=LB001 DEC=LB001
MOVL C00058 V=17 PL=LB000 ACC=LB001 DEC=LB001
MOVL C00059 V=7 PL=LB000 ACC=LB001 DEC=LB001
MOVL C00060 V=17 PL=LB000 ACC=LB001 DEC=LB001
MOVL C00061 V=17 PL=LB000 ACC=LB001 DEC=LB001
MOVL C00062 V=7 PL=LB000 ACC=LB001 DEC=LB001
MOVL C00063 V=17 PL=LB000 ACC=LB001 DEC=LB001
MOVL C00064 V=17 PL=LB000 ACC=LB001 DEC=LB001
MOVL C00065 V=7 PL=LB000 ACC=LB001 DEC=LB001
MOVL C00066 V=17 PL=LB000 ACC=LB001 DEC=LB001
MOVL C00067 V=17 PL=LB000 ACC=LB001 DEC=LB001
MOVL C00068 V=7 PL=LB000 ACC=LB001 DEC=LB001
MOVL C00069 V=17 PL=LB000 ACC=LB001 DEC=LB001
MOVL C00070 V=17 PL=LB000 ACC=LB001 DEC=LB001
MOVL C00071 V=7 PL=LB000 ACC=LB001 DEC=LB001
MOVL C00072 V=17 PL=LB000 ACC=LB001 DEC=LB001
MOVL C00073 V=17 PL=LB000 ACC=LB001 DEC=LB001
MOVL C00074 V=7 PL=LB000 ACC=LB001 DEC=LB001
MOVL C00075 V=17 PL=LB000 ACC=LB001 DEC=LB001
MOVL C00076 V=17 PL=LB000 ACC=LB001 DEC=LB001
MOVL C00077 V=7 PL=LB000 ACC=LB001 DEC=LB001
MOVL C00078 V=17 PL=LB000 ACC=LB001 DEC=LB001
MOVL C00079 V=17 PL=LB000 ACC=LB001 DEC=LB001
MOVL C00080 V=7 PL=LB000 ACC=LB001 DEC=LB001
MOVL C00081 V=17 PL=LB000 ACC=LB001 DEC=LB001
MOVL C00082 V=17 PL=LB000 ACC=LB001 DEC=LB001
MOVL C00083 V=7 PL=LB000 ACC=LB001 DEC=LB001
MOVL C00084 V=17 PL=LB000 ACC=LB001 DEC=LB001
MOVL C00085 V=17 PL=LB000 ACC=LB001 DEC=LB001
MOVL C00086 V=7 PL=LB000 ACC=LB001 DEC=LB001
MOVL C00087 V=17 PL=LB000 ACC=LB001 DEC=LB001
MOVL C00088 V=17 PL=LB000 ACC=LB001 DEC=LB001
MOVL C00089 V=7 PL=LB000 ACC=LB001 DEC=LB001
MOVL C00090 V=17 PL=LB000 ACC=LB001 DEC=LB001
MOVL C00091 V=17 PL=LB000 ACC=LB001 DEC=LB001
MOVL C00092 V=7 PL=LB000 ACC=LB001 DEC=LB001
MOVL C00093 V=17 PL=LB000 ACC=LB001 DEC=LB001
MOVL C00094 V=17 PL=LB000 ACC=LB001 DEC=LB001
MOVL C00095 V=7 PL=LB000 ACC=LB001 DEC=LB001
MOVL C00096 V=17 PL=LB000 ACC=LB001 DEC=LB001
MOVL C00097 V=17 PL=LB000 ACC=LB001 DEC=LB001
MOVL C00098 V=17 PL=LB000 ACC=LB001 DEC=LB001
MOVL C00099 V=17 PL=LB000 ACC=LB001 DEC=LB001
MOVL C00100 V=17 PL=LB000 ACC=LB001 DEC=LB001
MOVL C00101 V=7 PL=LB000 ACC=LB001 DEC=LB001
MOVL C00102 V=17 PL=LB000 ACC=LB001 DEC=LB001
MOVL C00103 V=17 PL=LB000 ACC=LB001 DEC=LB001
MOVL C00104 V=7 PL=LB000 ACC=LB001 DEC=LB001
MOVL C00105 V=17 PL=LB000 ACC=LB001 DEC=LB001
MOVL C00106 V=17 PL=LB000 ACC=LB001 DEC=LB001
MOVL C00107 V=7 PL=LB000 ACC=LB001 DEC=LB001
MOVL C00108 V=17 PL=LB000 ACC=LB001 DEC=LB001
MOVL C00109 V=17 PL=LB000 ACC=LB001 DEC=LB001
MOVL C00110 V=7 PL=LB000 ACC=LB001 DEC=LB001
MOVL C00111 V=17 PL=LB000 ACC=LB001 DEC=LB001
MOVL C00112 V=17 PL=LB000 ACC=LB001 DEC=LB001
MOVL C00113 V=7 PL=LB000 ACC=LB001 DEC=LB001
MOVL C00114 V=17 PL=LB000 ACC=LB001 DEC=LB001
MOVL C00115 V=17 PL=LB000 ACC=LB001 DEC=LB001
MOVL C00116 V=7 PL=LB000 ACC=LB001 DEC=LB001
MOVL C00117 V=17 PL=LB000 ACC=LB001 DEC=LB001
MOVL C00118 V=17 PL=LB000 ACC=LB001 DEC=LB001
MOVL C00119 V=7 PL=LB000 ACC=LB001 DEC=LB001
MOVL C00120 V=17 PL=LB000 ACC=LB001 DEC=LB001
MOVL C00121 V=17 PL=LB000 ACC=LB001 DEC=LB001
MOVL C00122 V=7 PL=LB000 ACC=LB001 DEC=LB001
MOVL C00123 V=17 PL=LB000 ACC=LB001 DEC=LB001
MOVL C00124 V=17 PL=LB000 ACC=LB001 DEC=LB001
MOVL C00125 V=7 PL=LB000 ACC=LB001 DEC=LB001
MOVL C00126 V=17 PL=LB000 ACC=LB001 DEC=LB001
MOVL C00127 V=17 PL=LB000 ACC=LB001 DEC=LB001
MOVL C00128 V=7 PL=LB000 ACC=LB001 DEC=LB001
MOVL C00129 V=17 PL=LB000 ACC=LB001 DEC=LB001
MOVL C00130 V=17 PL=LB000 ACC=LB001 DEC=LB001
MOVL C00131 V=7 PL=LB000 ACC=LB001 DEC=LB001
MOVL C00132 V=17 PL=LB000 ACC=LB001 DEC=LB001
MOVL C00133 V=17 PL=LB000 ACC=LB001 DEC=LB001
MOVL C00134 V=7 PL=LB000 ACC=LB001 DEC=LB001
MOVL C00135 V=17 PL=LB000 ACC=LB001 DEC=LB001
MOVL C00136 V=17 PL=LB000 ACC=LB001 DEC=LB001
MOVL C00137 V=7 PL=LB000 ACC=LB001 DEC=LB001
MOVL C00138 V=17 PL=LB000 ACC=LB001 DEC=LB001
MOVL C00139 V=17 PL=LB000 ACC=LB001 DEC=LB001
MOVL C00140 V=7 PL=LB000 ACC=LB001 DEC=LB001
MOVL C00141 V=17 PL=LB000 ACC=LB001 DEC=LB001
MOVL C00142 V=17 PL=LB000 ACC=LB001 DEC=LB001
MOVL C00143 V=7 PL=LB000 ACC=LB001 DEC=LB001
MOVL C00144 V=17 PL=LB000 ACC=LB001 DEC=LB001
MOVL C00145 V=17 PL=LB000 ACC=LB001 DEC=LB001
MOVL C00146 V=7 PL=LB000 ACC=LB001 DEC=LB001
MOVL C00147 V=17 PL=LB000 ACC=LB001 DEC=LB001
MOVL C00148 V=17 PL=LB000 ACC=LB001 DEC=LB001
MOVL C00149 V=7 PL=LB000 ACC=LB001 DEC=LB001
MOVL C00150 V=17 PL=LB000 ACC=LB001 DEC=LB001
MOVL C00151 V=17 PL=LB000 ACC=LB001 DEC=LB001
MOVL C00152 V=7 PL=LB000 ACC=LB001 DEC=LB001
MOVL C00153 V=17 PL=LB000 ACC=LB001 DEC=LB001
MOVL C00154 V=17 PL=LB000 ACC=LB001 DEC=LB001
MOVL C00155 V=7 PL=LB000 ACC=LB001 DEC=LB001
MOVL C00156 V=17 PL=LB000 ACC=LB001 DEC=LB001
MOVL C00157 V=17 PL=LB000 ACC=LB001 DEC=LB001
MOVL C00158 V=7 PL=LB000 ACC=LB001 DEC=LB001
MOVL C00159 V=17 PL=LB000 ACC=LB001 DEC=LB001
MOVL C00160 V=17 PL=LB000 ACC=LB001 DEC=LB001
MOVL C00161 V=7 PL=LB000 ACC=LB001 DEC=LB001
MOVL C00162 V=17 PL=LB000 ACC=LB001 DEC=LB001
MOVL C00163 V=17 PL=LB000 ACC=LB001 DEC=LB001
MOVL C00164 V=7 PL=LB000 ACC=LB001 DEC=LB001
MOVL C00165 V=17 PL=LB000 ACC=LB001 DEC=LB001
MOVL C00166 V=17 PL=LB000 ACC=LB001 DEC=LB001
MOVL C00167 V=7 PL=LB000 ACC=LB001 DEC=LB001
MOVL C00168 V=17 PL=LB000 ACC=LB001 DEC=LB001
MOVL C00169 V=17 PL=LB000 ACC=LB001 DEC=LB001
MOVL C00170 V=7 PL=LB000 ACC=LB001 DEC=LB001
MOVL C00171 V=17 PL=LB000 ACC=LB001 DEC=LB001
MOVL C00172 V=17 PL=LB000 ACC=LB001 DEC=LB001
MOVL C00173 V=7 PL=LB000 ACC=LB001 DEC=LB001
MOVL C00174 V=17 PL=LB000 ACC=LB001 DEC=LB001
MOVL C00175 V=17 PL=LB000 ACC=LB001 DEC=LB001
MOVL C00176 V=7 PL=LB000 ACC=LB001 DEC=LB001
MOVL C00177 V=17 PL=LB000 ACC=LB001 DEC=LB001
MOVL C00178 V=17 PL=LB000 ACC=LB001 DEC=LB001
MOVL C00179 V=7 PL=LB000 ACC=LB001 DEC=LB001
MOVL C00180 V=17 PL=LB000 ACC=LB001 DEC=LB001
MOVL C00181 V=17 PL=LB000 ACC=LB001 DEC=LB001
MOVL C00182 V=7 PL=LB000 ACC=LB001 DEC=LB001
MOVL C00183 V=17 PL=LB000 ACC=LB001 DEC=LB001
MOVL C00184 V=17 PL=LB000 ACC=LB001 DEC=LB001
MOVL C00185 V=7 PL=LB000 ACC=LB001 DEC=LB001
MOVL C00186 V=17 PL=LB000 ACC=LB001 DEC=LB001
MOVL C00187 V=17 PL=LB000 ACC=LB001 DEC=LB001
MOVL C00188 V=7 PL=LB000 ACC=LB001 DEC=LB001
MOVL C00189 V=17 PL=LB000 ACC=LB001 DEC=LB001
MOVL C00190 V=17 PL=LB000 ACC=LB001 DEC=LB001
MOVL C00191 V=7 PL=LB000 ACC=LB001 DEC=LB001
MOVL C00192 V=17 PL=LB000 ACC=LB001 DEC=LB001
' Rapid Move Starts
MOVL C00193 V=17 PL=LB000 ACC=LB001 DEC=LB001
' By Autodesk Fusion CAM 2.0.20494
' Tool = 3
' Spindle = 5000 RPM
' Set Position Level
' Set Acceleration
' Program Start
' First Toolpath Point
END
